TYPE FsST_PlcTaskInformation EXTENDS PlcTaskSystemInfo :
STRUCT
	CycleTicks : LTIME; // Current task cycle time
END_STRUCT
END_TYPE

(* stored: Version 1.1.0.1, ProductVersion 3.1.4024.4
   DUT FsST_PlcTaskInformation: Id {311720c0-a47e-4a31-a1d4-f7cf7324c3a4} *)
